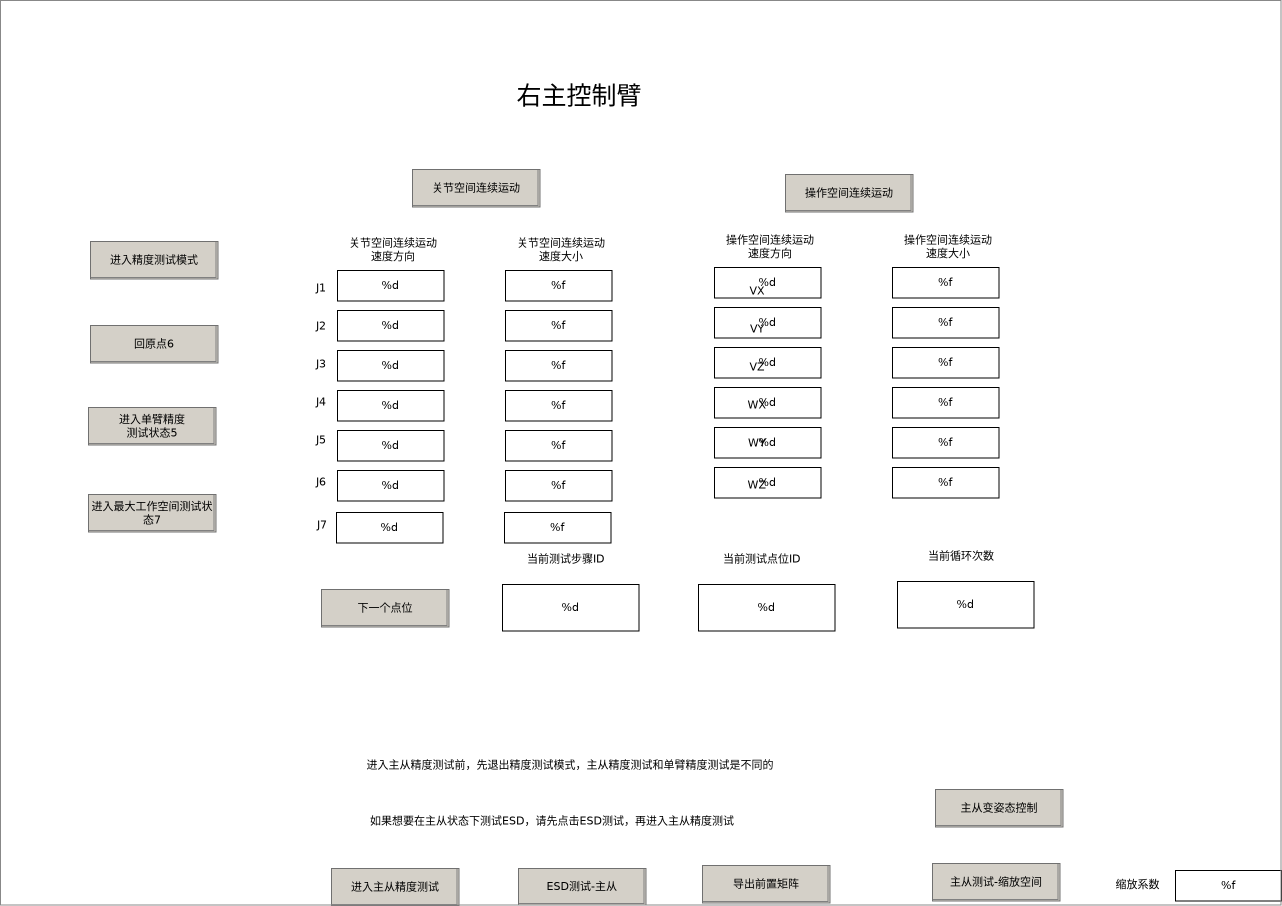
VISUALIZATION precision_a2  // 1282x906
    Label (504,74 150x43), "右主控制臂"
    Rectangle (337,270 107x31), "%d", text variable: g_motionTest.m_jntMotionDir[2][1]
        OnMouseClick: write the text variable via Default, min -1, max 1
    Label (318,235 150x29), "关节空间连续运动 速度方向"
    Rectangle (337,310 107x31), "%d", text variable: g_motionTest.m_jntMotionDir[2][2]
        OnMouseClick: write the text variable via Default, min -1, max 1
    Rectangle (337,350 107x31), "%d", text variable: g_motionTest.m_jntMotionDir[2][3]
        OnMouseClick: write the text variable via Default, min -1, max 1
    Rectangle (337,390 107x31), "%d", text variable: g_motionTest.m_jntMotionDir[2][4]
        OnMouseClick: write the text variable via Default, min -1, max 1
    Rectangle (337,430 107x31), "%d", text variable: g_motionTest.m_jntMotionDir[2][5]
        OnMouseClick: write the text variable via Default, min -1, max 1
    Rectangle (337,470 107x31), "%d", text variable: g_motionTest.m_jntMotionDir[2][6]
        OnMouseClick: write the text variable via Default, min -1, max 1
    Rectangle (505,270 107x31), "%f", text variable: g_motionTest.m_jntVel[2][1]
        OnMouseClick: write the text variable via Default
    Label (486,235 150x29), "关节空间连续运动 速度大小"
    Rectangle (505,310 107x31), "%f", text variable: g_motionTest.m_jntVel[2][2]
        OnMouseClick: write the text variable via Default
    Rectangle (505,350 107x31), "%f", text variable: g_motionTest.m_jntVel[2][3]
        OnMouseClick: write the text variable via Default
    Rectangle (505,390 107x31), "%f", text variable: g_motionTest.m_jntVel[2][4]
        OnMouseClick: write the text variable via Default
    Rectangle (505,430 107x31), "%f", text variable: g_motionTest.m_jntVel[2][5]
        OnMouseClick: write the text variable via Default
    Rectangle (505,470 107x31), "%f", text variable: g_motionTest.m_jntVel[2][6]
        OnMouseClick: write the text variable via Default
    Rectangle (714,267 107x31), "%d", text variable: g_motionTest.m_spatialMotionDir[2][1]
        OnMouseClick: write the text variable via Default, min -1, max 1
    Label (695,232 150x29), "操作空间连续运动 速度方向"
    Rectangle (714,307 107x31), "%d", text variable: g_motionTest.m_spatialMotionDir[2][2]
        OnMouseClick: write the text variable via Default, min -1, max 1
    Rectangle (714,347 107x31), "%d", text variable: g_motionTest.m_spatialMotionDir[2][3]
        OnMouseClick: write the text variable via Default, min -1, max 1
    Rectangle (714,387 107x31), "%d", text variable: g_motionTest.m_spatialMotionDir[2][4]
        OnMouseClick: write the text variable via Default, min -1, max 1
    Rectangle (714,427 107x31), "%d", text variable: g_motionTest.m_spatialMotionDir[2][5]
        OnMouseClick: write the text variable via Default, min -1, max 1
    Rectangle (714,467 107x31), "%d", text variable: g_motionTest.m_spatialMotionDir[2][6]
        OnMouseClick: write the text variable via Default, min -1, max 1
    Rectangle (892,267 107x31), "%f", text variable: g_motionTest.m_spatialVel[2][1]
        OnMouseClick: write the text variable via Default
    Label (873,232 150x29), "操作空间连续运动 速度大小"
    Rectangle (892,307 107x31), "%f", text variable: g_motionTest.m_spatialVel[2][2]
        OnMouseClick: write the text variable via Default
    Rectangle (892,347 107x31), "%f", text variable: g_motionTest.m_spatialVel[2][3]
        OnMouseClick: write the text variable via Default
    Rectangle (892,387 107x31), "%f", text variable: g_motionTest.m_spatialVel[2][4]
        OnMouseClick: write the text variable via Default
    Rectangle (892,427 107x31), "%f", text variable: g_motionTest.m_spatialVel[2][5]
        OnMouseClick: write the text variable via Default
    Rectangle (892,467 107x31), "%f", text variable: g_motionTest.m_spatialVel[2][6]
        OnMouseClick: write the text variable via Default
    Button (90,241 128x38), "进入精度测试模式", colour toggle: g_motionTest.m_enterPrecisionTestMode[2]
        toggle g_motionTest.m_enterPrecisionTestMode[2]
    Button (412,169 128x38), "关节空间连续运动", colour toggle: g_motionTest.m_uiArmModeL[2,2]
        tap g_motionTest.m_uiArmMode[2,2]
    Button (785,174 128x38), "操作空间连续运动", colour toggle: g_motionTest.m_uiArmModeL[2,4]
        tap g_motionTest.m_uiArmMode[2,4]
    Button (90,325 128x38), "回原点6", colour toggle: g_motionTest.m_uiArmModeL[2,6]
        tap g_motionTest.m_uiArmMode[2,6]
    Button (321,589 128x38), "下一个点位", colour toggle: g_motionTest.m_nextStep[2]
        tap g_motionTest.m_nextStep[2]
    Group (491,541 545x90)
        Rectangle (11,43 137x47), "%d", text variable: g_motionTest.m_curStep[2]
        Label (0,3 150x30), "当前测试步骤ID"
        Rectangle (207,43 137x47), "%d", text variable: g_motionTest.m_testPointId[2]
        Label (196,3 150x30), "当前测试点位ID"
        Rectangle (406,40 137x47), "%d", text variable: g_motionTest.m_testCycleId[2]
        Label (395,0 150x30), "当前循环次数"
    Group (314,273 14x224)
        Label (0,0 14x30), "J1"
        Label (0,38 14x30), "J2"
        Label (0,76 14x30), "J3"
        Label (0,114 14x30), "J4"
        Label (0,152 14x30), "J5"
        Label (0,194 14x30), "J6"
    Group (682,276 26x224)
        Label (0,0 150x30), "VX"
        Label (0,38 150x30), "VY"
        Label (0,76 150x30), "VZ"
        Label (0,114 150x30), "WX"
        Label (0,152 150x30), "WY"
        Label (0,194 150x30), "WZ"
    Button (88,407 128x38), "进入单臂精度 测试状态5", colour toggle: g_motionTest.m_uiArmModeL[2,5]
        toggle g_motionTest.m_uiArmMode[2,5]
    Button (88,494 128x38), "进入最大工作空间测试状态7", colour toggle: g_motionTest.m_uiArmModeL[2,7]
        toggle g_motionTest.m_uiArmMode[2,7]
    Button (331,868 128x38), "进入主从精度测试", colour toggle: g_motionTest.m_MSPrecisionTest[2]
        toggle g_motionTest.m_MSPrecisionTest[2]
    Label (315,510 14x30), "J7"
    Rectangle (336,512 107x31), "%d", text variable: g_motionTest.m_jntMotionDir[2][7]
        OnMouseClick: write the text variable via Default, min -1, max 1
    Rectangle (504,512 107x31), "%f", text variable: g_motionTest.m_jntVel[2][7]
        OnMouseClick: write the text variable via Default
    Button (702,865 128x38), "导出前置矩阵"
        tap g_motionTest.m_writeData[2]
    Button (518,868 128x37), "ESD测试-主从", colour toggle: g_motionTest.m_esdTest[2]
        toggle g_motionTest.m_esdTest[2]
    Label (251,750 638x30), "进入主从精度测试前，先退出精度测试模式，主从精度测试和单臂精度测试是不同的"
    Label (233,806 638x30), "如果想要在主从状态下测试ESD，请先点击ESD测试，再进入主从精度测试"
    Button (935,789 128x38), "主从变姿态控制", colour toggle: g_motionTest.m_poseChange
        toggle g_motionTest.m_poseChange
    Button (932,863 128x38), "主从测试-缩放空间", colour toggle: g_motionTest.m_scaleSpace
        toggle g_motionTest.m_scaleSpace
    Rectangle (1175,870 107x31), "%f", text variable: GVL_Const.g_scaleFactor
        OnMouseClick: write the text variable via Default
    Label (1088,868 99x33), "缩放系数"
END_VISUALIZATION

(* stored: Version 1.1.0.1, ProductVersion 3.1.4024.11
   Visu precision_a2: Id {74e91e78-0d55-4701-a331-76ce179a9c2d} *)
